FUNCTION_BLOCK E_RENDXTRM (* Basic Function Block Type *)
  (* Standard: 61499-2 *)
  (* Version 0.0, 2015-11-13, 4DIAC-IDE, 4DIAC-Consortium *)
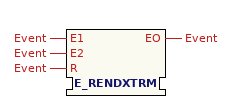
  EVENT_INPUT
    E1; (* Initialization Request *)
    E2; (* Normal Execution Request *)
    R;
  END_EVENT
  EVENT_OUTPUT
    EO; (* Execution Confirmation *)
  END_EVENT
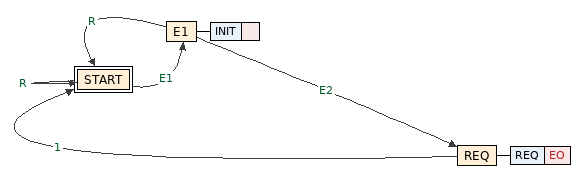
  EC_STATES
    START; (* Initial State *)
    E1 : INIT; (* Initialization *)
    REQ : REQ -> EO; (* Normal execution *)
  END_STATES
  EC_TRANSITIONS
    START TO E1 := E1;
    E1 TO START := R;
    REQ TO START := 1;
    E1 TO REQ := E2;
    START TO START := R;
  END_TRANSITIONS
  ALGORITHM INIT IN ST: (* Initialization algorithm *)

  END_ALGORITHM
  ALGORITHM REQ IN ST: (* Normally executed algorithm *)

  END_ALGORITHM
END_FUNCTION_BLOCK
